PROGRAM Datos_Caudalimetros
VAR
END_VAR

(*
HMI.CA1_L1_FT1_caudal	:= SEL(TO_REAL(Entradas.CA1_L1_FT1_caudal.icaudal)*16.6667/1000 > 0, 0, TO_REAL(Entradas.CA1_L1_FT1_caudal.icaudal)*16.6667/1000);		// Em L/min 
HMI.CA1_L1_FT1_temp 	:= TO_REAL(Entradas.CA1_L1_FT1_temp.itemp)*0.01; // en grados centigrados
HMI.CA1_L2_FT1_caudal	:= SEL(TO_REAL(Entradas.CA1_L2_FT1_caudal.icaudal)*16.6667/1000 > 0, 0, TO_REAL(Entradas.CA1_L2_FT1_caudal.icaudal)*16.6667/1000);		// Em L/min 
HMI.CA1_L2_FT1_temp		:= TO_REAL(Entradas.CA1_L2_FT1_temp.itemp)*0.01; // en grados centigrados
HMI.CA1_L3_FT1_caudal 	:= SEL(TO_REAL(Entradas.CA1_L3_FT1_caudal.icaudal)*16.6667/1000 > 0, 0, TO_REAL(Entradas.CA1_L3_FT1_caudal.icaudal)*16.6667/1000);		// Em L/min
HMI.CA1_L3_FT1_temp 	:= TO_REAL(Entradas.CA1_L3_FT1_temp.itemp)*0.01; // en grados centigrados
HMI.CA1_L4_FT1_caudal 	:= SEL(TO_REAL(Entradas.CA1_L4_FT1_caudal.icaudal)*16.6667/1000 > 0, 0, TO_REAL(Entradas.CA1_L4_FT1_caudal.icaudal)*16.6667/1000);		// Em L/min
HMI.CA1_L4_FT1_temp 	:= TO_REAL(Entradas.CA1_L4_FT1_temp.itemp)*0.01; // en grados centigrados
HMI.CA2_L5_FT1_caudal 	:= SEL(TO_REAL(Entradas.CA2_L5_FT1_caudal.icaudal)*16.6667/1000 > 0, 0, TO_REAL(Entradas.CA2_L5_FT1_caudal.icaudal)*16.6667/1000);		// Em L/min
HMI.CA2_L5_FT1_temp 	:= TO_REAL(Entradas.CA2_L5_FT1_temp.itemp)*0.01; // en grados centigrados
HMI.CA2_L6_FT1_caudal 	:= SEL(TO_REAL(Entradas.CA2_L6_FT1_caudal.icaudal)*16.6667/1000 > 0, 0, TO_REAL(Entradas.CA2_L6_FT1_caudal.icaudal)*16.6667/1000);		// Em L/min
HMI.CA2_L6_FT1_temp 	:= TO_REAL(Entradas.CA2_L6_FT1_temp.itemp)*0.01; // en grados centigrados
HMI.CA2_L7_FT1_caudal 	:= SEL(TO_REAL(Entradas.CA2_L7_FT1_caudal.icaudal)*16.6667/1000 > 0, 0, TO_REAL(Entradas.CA2_L7_FT1_caudal.icaudal)*16.6667/1000);		// Em L/min
HMI.CA2_L7_FT1_temp 	:= TO_REAL(Entradas.CA2_L7_FT1_temp.itemp)*0.01; // en grados centigrados
HMI.CA2_L8_FT1_caudal 	:= SEL(TO_REAL(Entradas.CA2_L8_FT1_caudal.icaudal)*16.6667/1000 > 0, 0, TO_REAL(Entradas.CA2_L8_FT1_caudal.icaudal)*16.6667/1000);		// Em L/min
HMI.CA2_L8_FT1_temp 	:= TO_REAL(Entradas.CA2_L8_FT1_temp.itemp)*0.01; // en grados centigrados
HMI.CA3_L9_FT1_caudal 	:= SEL(TO_REAL(Entradas.CA3_L9_FT1_caudal.icaudal)*16.6667/1000 > 0, 0, TO_REAL(Entradas.CA3_L9_FT1_caudal.icaudal)*16.6667/1000);		// Em L/min
HMI.CA3_L9_FT1_temp 	:= TO_REAL(Entradas.CA3_L9_FT1_temp.itemp)*0.01; // en grados centigrados
HMI.CA3_L10_FT1_caudal 	:= SEL(TO_REAL(Entradas.CA3_L10_FT1_caudal.icaudal)*16.6667/1000 > 0, 0, TO_REAL(Entradas.CA3_L10_FT1_caudal.icaudal)*16.6667/1000);		// Em L/min
HMI.CA3_L10_FT1_temp 	:= TO_REAL(Entradas.CA3_L10_FT1_temp.itemp)*0.01; // en grados centigrados
HMI.CA3_L11_FT1_caudal 	:= SEL(TO_REAL(Entradas.CA3_L11_FT1_caudal.icaudal)*16.6667/1000 > 0, 0, TO_REAL(Entradas.CA3_L11_FT1_caudal.icaudal)*16.6667/1000);		// Em L/min
HMI.CA3_L11_FT1_temp 	:= TO_REAL(Entradas.CA3_L11_FT1_temp.itemp)*0.01; // en grados centigrados 
HMI.CA3_L12_FT1_caudal 	:= SEL(TO_REAL(Entradas.CA3_L12_FT1_caudal.icaudal)*16.6667/1000 > 0, 0, TO_REAL(Entradas.CA3_L12_FT1_caudal.icaudal)*16.6667/1000);		// Em L/min
HMI.CA3_L12_FT1_temp 	:= TO_REAL(Entradas.CA3_L12_FT1_temp.itemp)*0.01; // en grados centigrados
//
HMI.TR_L1_FT2_caudal	:= SEL(TO_REAL(Entradas.TR_L1_FT2_caudal.icaudal)*16.6667/1000 > 0, 0, TO_REAL(Entradas.TR_L1_FT2_caudal.icaudal)*16.6667/1000); // en ml/s
HMI.TR_L1_FT2_temp 		:= TO_REAL(Entradas.TR_L1_FT2_temp.itemp)*0.01; // en grados centigrados
HMI.TR_L2_FT2_caudal 	:= SEL(TO_REAL(Entradas.TR_L2_FT2_caudal.icaudal)*16.6667/1000 > 0, 0, TO_REAL(Entradas.TR_L2_FT2_caudal.icaudal)*16.6667/1000); // en ml/s
HMI.TR_L2_FT2_temp 		:= TO_REAL(Entradas.TR_L2_FT2_temp.itemp)*0.01; // en grados centigrados
HMI.TR_L3_FT2_caudal 	:= SEL(TO_REAL(Entradas.TR_L3_FT2_caudal.icaudal)*16.6667/1000 > 0, 0, TO_REAL(Entradas.TR_L3_FT2_caudal.icaudal)*16.6667/1000); // en ml/s
HMI.TR_L3_FT2_temp 		:= TO_REAL(Entradas.TR_L3_FT2_temp.itemp)*0.01; // en grados centigrados
HMI.TR_L4_FT2_caudal 	:= SEL(TO_REAL(Entradas.TR_L4_FT2_caudal.icaudal)*16.6667/1000 > 0, 0, TO_REAL(Entradas.TR_L4_FT2_caudal.icaudal)*16.6667/1000); // en ml/s
HMI.TR_L4_FT2_temp 		:= TO_REAL(Entradas.TR_L4_FT2_temp.itemp)*0.01; // en grados centigrados
HMI.TR_L5_FT2_caudal 	:= SEL(TO_REAL(Entradas.TR_L5_FT2_caudal.icaudal)*16.6667/1000 > 0, 0, TO_REAL(Entradas.TR_L5_FT2_caudal.icaudal)*16.6667/1000); // en ml/s
HMI.TR_L5_FT2_temp 		:= TO_REAL(Entradas.TR_L5_FT2_temp.itemp)*0.01; // en grados centigrados
HMI.TR_L6_FT2_caudal 	:= SEL(TO_REAL(Entradas.TR_L6_FT2_caudal.icaudal)*16.6667/1000 > 0, 0, TO_REAL(Entradas.TR_L6_FT2_caudal.icaudal)*16.6667/1000); // en ml/s
HMI.TR_L6_FT2_temp 		:= TO_REAL(Entradas.TR_L6_FT2_temp.itemp)*0.01; // en grados centigrados
HMI.TR_L7_FT2_caudal 	:= SEL(TO_REAL(Entradas.TR_L7_FT2_caudal.icaudal)*16.6667/1000 > 0, 0, TO_REAL(Entradas.TR_L7_FT2_caudal.icaudal)*16.6667/1000); // en ml/s
HMI.TR_L7_FT2_temp 		:= TO_REAL(Entradas.TR_L7_FT2_temp.itemp)*0.01; // en grados centigrados
HMI.TR_L8_FT2_caudal 	:= SEL(TO_REAL(Entradas.TR_L8_FT2_caudal.icaudal)*16.6667/1000 > 0, 0, TO_REAL(Entradas.TR_L8_FT2_caudal.icaudal)*16.6667/1000); // en ml/s
HMI.TR_L8_FT2_temp 		:= TO_REAL(Entradas.TR_L8_FT2_temp.itemp)*0.01; // en grados centigrados
HMI.TR_L9_FT2_caudal 	:= SEL(TO_REAL(Entradas.TR_L9_FT2_caudal.icaudal)*16.6667/1000 > 0, 0, TO_REAL(Entradas.TR_L9_FT2_caudal.icaudal)*16.6667/1000); // en ml/s
HMI.TR_L9_FT2_temp 		:= TO_REAL(Entradas.TR_L9_FT2_temp.itemp)*0.01; // en grados centigrados
HMI.TR_L10_FT2_caudal 	:= SEL(TO_REAL(Entradas.TR_L10_FT2_caudal.icaudal)*16.6667/1000 > 0, 0, TO_REAL(Entradas.TR_L10_FT2_caudal.icaudal)*16.6667/1000); // en ml/s
HMI.TR_L10_FT2_temp 	:= TO_REAL(Entradas.TR_L10_FT2_temp.itemp)*0.01; // en grados centigrados
HMI.TR_L11_FT2_caudal 	:= SEL(TO_REAL(Entradas.TR_L11_FT2_caudal.icaudal)*16.6667/1000 > 0, 0, TO_REAL(Entradas.TR_L11_FT2_caudal.icaudal)*16.6667/1000); // en ml/s
HMI.TR_L11_FT2_temp 	:= TO_REAL(Entradas.TR_L11_FT2_temp.itemp)*0.01; // en grados centigrados
HMI.TR_L12_FT2_caudal 	:= SEL(TO_REAL(Entradas.TR_L12_FT2_caudal.icaudal)*16.6667/1000 > 0, 0, TO_REAL(Entradas.TR_L12_FT2_caudal.icaudal)*16.6667/1000); // en ml/s
HMI.TR_L12_FT2_temp 	:= TO_REAL(Entradas.TR_L12_FT2_temp.itemp)*0.01; // en grados centigrados

*)

{Region "Sensores dos totens"}

//Sensores de vazão doos totens
	HMI.CA1_L1_FT1_caudal	:=TO_REAL(Entradas.CA1_L1_FT1_caudal.icaudal)*0.0166667*16.6667; // en ml/s
	HMI.CA1_L2_FT1_caudal	:=TO_REAL(Entradas.CA1_L2_FT1_caudal.icaudal)*0.0166667*16.6667; // en ml/s
	HMI.CA1_L3_FT1_caudal	:=TO_REAL(Entradas.CA1_L3_FT1_caudal.icaudal)*0.0166667*16.6667; // en ml/s
	HMI.CA1_L4_FT1_caudal 	:=TO_REAL(Entradas.CA1_L4_FT1_caudal.icaudal)*0.0166667*16.6667; // en ml/s
	HMI.CA2_L5_FT1_caudal 	:=TO_REAL(Entradas.CA2_L5_FT1_caudal.icaudal)*0.0166667*16.6667; // en ml/s
	HMI.CA2_L6_FT1_caudal 	:=TO_REAL(Entradas.CA2_L6_FT1_caudal.icaudal)*0.0166667*16.6667; // en ml/s
	HMI.CA2_L7_FT1_caudal 	:=TO_REAL(Entradas.CA2_L7_FT1_caudal.icaudal)*0.0166667*16.6667; // en ml/s
	HMI.CA2_L8_FT1_caudal 	:=TO_REAL(Entradas.CA2_L8_FT1_caudal.icaudal)*0.0166667*16.6667; // en ml/s
	HMI.CA3_L9_FT1_caudal 	:=TO_REAL(Entradas.CA3_L9_FT1_caudal.icaudal)*0.0166667*16.6667; // en ml/s
	HMI.CA3_L10_FT1_caudal 	:=TO_REAL(Entradas.CA3_L10_FT1_caudal.icaudal)*0.0166667*16.6667; // en ml/s
	HMI.CA3_L11_FT1_caudal 	:=TO_REAL(Entradas.CA3_L11_FT1_caudal.icaudal)*0.00166667*16.6667; // en ml/s
	HMI.CA3_L12_FT1_caudal 	:=TO_REAL(Entradas.CA3_L12_FT1_caudal.icaudal)*0.00166667*16.6667; // en ml/s
	
	//Sensores de temperatura dos totens
	HMI.CA1_L1_FT1_temp		:=TO_REAL(Entradas.CA1_L1_FT1_temp.itemp)*0.01; // en grados centigrados
	HMI.CA1_L2_FT1_temp		:=TO_REAL(Entradas.CA1_L2_FT1_temp.itemp)*0.01; // en grados centigrados
	HMI.CA1_L3_FT1_temp 	:=TO_REAL(Entradas.CA1_L3_FT1_temp.itemp)*0.01; // en grados centigrados
	HMI.CA1_L4_FT1_temp 	:=TO_REAL(Entradas.CA1_L4_FT1_temp.itemp)*0.01; // en grados centigrados
	HMI.CA2_L5_FT1_temp 	:=TO_REAL(Entradas.CA2_L5_FT1_temp.itemp)*0.01; // en grados centigrados
	HMI.CA2_L6_FT1_temp 	:=TO_REAL(Entradas.CA2_L6_FT1_temp.itemp)*0.01; // en grados centigrados
	HMI.CA2_L7_FT1_temp 	:=TO_REAL(Entradas.CA2_L7_FT1_temp.itemp)*0.01; // en grados centigrados
	HMI.CA2_L8_FT1_temp 	:=TO_REAL(Entradas.CA2_L8_FT1_temp.itemp)*0.01; // en grados centigrados
	HMI.CA3_L9_FT1_temp 	:=TO_REAL(Entradas.CA3_L9_FT1_temp.itemp)*0.01; // en grados centigrados
	HMI.CA3_L10_FT1_temp 	:=TO_REAL(Entradas.CA3_L10_FT1_temp.itemp)*0.01; // en grados centigrados
	HMI.CA3_L11_FT1_temp 	:=TO_REAL(Entradas.CA3_L11_FT1_temp.itemp)*0.01; // en grados centigrados
	HMI.CA3_L12_FT1_temp 	:=TO_REAL(Entradas.CA3_L12_FT1_temp.itemp)*0.01; // en grados centigrados
{endregion}


{Region "Sensores da tratadora"}

	//Sensores de vazão da tratadora
	HMI.TR_L1_FT2_caudal :=TO_REAL(Entradas.TR_L1_FT2_caudal.icaudal)*0.0166667*16.6667; // en ml/s
	HMI.TR_L2_FT2_caudal :=TO_REAL(Entradas.TR_L2_FT2_caudal.icaudal)*0.0166667*16.6667; // en ml/s
	HMI.TR_L3_FT2_caudal :=TO_REAL(Entradas.TR_L3_FT2_caudal.icaudal)*0.0166667*16.6667; // en ml/s
	HMI.TR_L4_FT2_caudal :=TO_REAL(Entradas.TR_L4_FT2_caudal.icaudal)*0.0166667*16.6667; // en ml/s
	HMI.TR_L5_FT2_caudal :=TO_REAL(Entradas.TR_L5_FT2_caudal.icaudal)*0.0166667*16.6667; // en ml/s
	HMI.TR_L6_FT2_caudal :=TO_REAL(Entradas.TR_L6_FT2_caudal.icaudal)*0.0166667*16.6667; // en ml/s
	HMI.TR_L7_FT2_caudal :=TO_REAL(Entradas.TR_L7_FT2_caudal.icaudal)*0.0166667*16.6667; // en ml/s
	HMI.TR_L8_FT2_caudal :=TO_REAL(Entradas.TR_L8_FT2_caudal.icaudal)*0.0166667*16.6667; // en ml/s
	HMI.TR_L9_FT2_caudal :=TO_REAL(Entradas.TR_L9_FT2_caudal.icaudal)*0.0166667*16.6667; // en ml/s
	HMI.TR_L10_FT2_caudal :=TO_REAL(Entradas.TR_L10_FT2_caudal.icaudal)*0.0166667*16.6667; // en ml/s
	HMI.TR_L11_FT2_caudal :=TO_REAL(Entradas.TR_L11_FT2_caudal.icaudal)*0.00166667*16.6667; // en ml/s
	HMI.TR_L12_FT2_caudal :=TO_REAL(Entradas.TR_L12_FT2_caudal.icaudal)*0.00166667*16.6667; // en ml/s
	
	//Sensores de temperatura da tratadora
	HMI.TR_L1_FT2_temp :=TO_REAL(Entradas.TR_L1_FT2_temp.itemp)*0.01; // en grados centigrados
	HMI.TR_L2_FT2_temp :=TO_REAL(Entradas.TR_L2_FT2_temp.itemp)*0.01; // en grados centigrados
	HMI.TR_L3_FT2_temp :=TO_REAL(Entradas.TR_L3_FT2_temp.itemp)*0.01; // en grados centigrados
	HMI.TR_L4_FT2_temp :=TO_REAL(Entradas.TR_L4_FT2_temp.itemp)*0.01; // en grados centigrados
	HMI.TR_L5_FT2_temp :=TO_REAL(Entradas.TR_L5_FT2_temp.itemp)*0.01; // en grados centigrados
	HMI.TR_L6_FT2_temp :=TO_REAL(Entradas.TR_L6_FT2_temp.itemp)*0.01; // en grados centigrados
	HMI.TR_L7_FT2_temp :=TO_REAL(Entradas.TR_L7_FT2_temp.itemp)*0.01; // en grados centigrados
	HMI.TR_L8_FT2_temp :=TO_REAL(Entradas.TR_L8_FT2_temp.itemp)*0.01; // en grados centigrados
	HMI.TR_L9_FT2_temp :=TO_REAL(Entradas.TR_L9_FT2_temp.itemp)*0.01; // en grados centigrados
	HMI.TR_L10_FT2_temp :=TO_REAL(Entradas.TR_L10_FT2_temp.itemp)*0.01; // en grados centigrados
	HMI.TR_L11_FT2_temp :=TO_REAL(Entradas.TR_L11_FT2_temp.itemp)*0.01; // en grados centigrados
	HMI.TR_L12_FT2_temp :=TO_REAL(Entradas.TR_L12_FT2_temp.itemp)*0.01;  // en grados centigrados

{endregion}

END_PROGRAM

(* stored: Version 1.1.0.1, ProductVersion 3.1.4024.14
   POU Datos_Caudalimetros: Id {5be0e032-cd28-443d-ba62-025f995b96b0}, SpecialFunc None *)
